{attribute 'GeneratedUsingTerminal: EL9222-4433-0018'}
{attribute addProperty BoxType "EL9222-4433-0018"}
{attribute addProperty Id "EtcSlaveTerminalBaseOCP_Inputs_Channel_1AT %I*OCP_Inputs_Channel_8CCE65FB11OCP_Inputs_Channel_2AT %I*OCP_Inputs_Channel_8CCE65FB11OCP_Outputs_Channel_1AT %Q*OCP_Outputs_Channel_010149342OCP_Outputs_Channel_2AT %Q*OCP_Outputs_Channel_010149342WcStateAT %I*WcState_9091E0EB2InfoDataAT %I*InfoData_32EB74EA10"}
{attribute addProperty CRC "74283812"}
{attribute addProperty Size "38"}
TYPE EL9222_046D7B24 EXTENDS EtcSlaveTerminalBase :
STRUCT
	{attribute addProperty Name "OCP_Inputs_Channel_1"}
	OCP_Inputs_Channel_1 : OCP_Inputs_Channel_8CCE65FB;
	{attribute addProperty Name "OCP_Inputs_Channel_2"}
	OCP_Inputs_Channel_2 : OCP_Inputs_Channel_8CCE65FB;
	{attribute addProperty Name "OCP_Outputs_Channel_1"}
	OCP_Outputs_Channel_1 : OCP_Outputs_Channel_01014934;
	{attribute addProperty Name "OCP_Outputs_Channel_2"}
	OCP_Outputs_Channel_2 : OCP_Outputs_Channel_01014934;
	{attribute addProperty Name "WcState"}
	WcState : WcState_9091E0EB;
	{attribute addProperty Name "InfoData"}
	InfoData : InfoData_32EB74EA;
END_STRUCT
END_TYPE

(* stored: Version 1.2.0.0, ProductVersion 3.1.4024.9
   DUT EL9222_046D7B24: Id {ec37c04f-d685-4475-8370-e98f9de45b91} *)
